FUNCTION_BLOCK FB_ProfidriveGSM_Test EXTENDS TcUnit.FB_TestSuite

TestState_S0();
TestState_S1();
TestState_S2();
TestState_S3();
TestState_S4();
TestState_S51();
TestState_S52();

TestTransitions_S0();
TestTransitions_S1();
TestTransitions_S2();
TestTransitions_S3();
TestTransitions_S4();
TestTransitions_S51();
TestTransitions_S52();

METHOD TestState_S0 : BOOL
VAR
	fbFSM 				: FB_ProfidriveGSM;
	stStatusExpected	: ST_ProfidriveGSM_Status;
END_VAR
TEST('Set State S0');

//Arrange
fbFSM.eState := E_ProfidriveGSM_State.S0_Disabled;

stStatusExpected.b0_ReadyToSwitchOn 		:= FALSE;				
stStatusExpected.b1_ReadyForOperation 		:= FALSE;				
stStatusExpected.b2_OperationEnabled 		:= FALSE;
stStatusExpected.b6_SwitchingOnInhibited 	:= FALSE;

//Act
fbFSM();

//Assert

AssertEquals_BOOL(stStatusExpected.b0_ReadyToSwitchOn, fbFSM.nStatus.b0_ReadyToSwitchOn, 'b0_ReadyToSwitchOn: AssertEquals not returning expected value');
AssertEquals_BOOL(stStatusExpected.b1_ReadyForOperation, fbFSM.nStatus.b1_ReadyForOperation, 'b1_ReadyForOperation: AssertEquals not returning expected value');
AssertEquals_BOOL(stStatusExpected.b2_OperationEnabled, fbFSM.nStatus.b2_OperationEnabled, 'b2_OperationEnabled: AssertEquals not returning expected value');	
AssertEquals_BOOL(stStatusExpected.b6_SwitchingOnInhibited, fbFSM.nStatus.b6_SwitchingOnInhibited, 'b6_SwitchingOnInhibited: AssertEquals not returning expected value');	

TEST_FINISHED();
END_METHOD

METHOD TestState_S1 : BOOL
VAR
	fbFSM 				: FB_ProfidriveGSM;
	stStatusExpected	: ST_ProfidriveGSM_Status;
END_VAR
TEST('Set State S1');

//Arrange
fbFSM.eState := E_ProfidriveGSM_State.S1_SwitchingOnInhibited;

stStatusExpected.b0_ReadyToSwitchOn 		:= FALSE;				
stStatusExpected.b1_ReadyForOperation 		:= FALSE;				
stStatusExpected.b2_OperationEnabled 		:= FALSE;
stStatusExpected.b6_SwitchingOnInhibited 	:= TRUE;

//Act
fbFSM();

//Assert
AssertEquals_BOOL(stStatusExpected.b0_ReadyToSwitchOn, fbFSM.nStatus.b0_ReadyToSwitchOn, 'b0_ReadyToSwitchOn: AssertEquals not returning expected value');
AssertEquals_BOOL(stStatusExpected.b1_ReadyForOperation, fbFSM.nStatus.b1_ReadyForOperation, 'b1_ReadyForOperation: AssertEquals not returning expected value');
AssertEquals_BOOL(stStatusExpected.b2_OperationEnabled, fbFSM.nStatus.b2_OperationEnabled, 'b2_OperationEnabled: AssertEquals not returning expected value');	
AssertEquals_BOOL(stStatusExpected.b6_SwitchingOnInhibited, fbFSM.nStatus.b6_SwitchingOnInhibited, 'b6_SwitchingOnInhibited: AssertEquals not returning expected value');	

TEST_FINISHED();
END_METHOD

METHOD TestState_S2 : BOOL
VAR
	fbFSM 				: FB_ProfidriveGSM;
	stStatusExpected	: ST_ProfidriveGSM_Status;
END_VAR
TEST('Set State S2');

//Arrange
fbFSM.eState := E_ProfidriveGSM_State.S2_ReadyForSwitchingOn;

stStatusExpected.b0_ReadyToSwitchOn 		:= TRUE;				
stStatusExpected.b1_ReadyForOperation 		:= FALSE;				
stStatusExpected.b2_OperationEnabled 		:= FALSE;
stStatusExpected.b6_SwitchingOnInhibited 	:= FALSE;

//Act
fbFSM();

//Assert
AssertEquals_BOOL(stStatusExpected.b0_ReadyToSwitchOn, fbFSM.nStatus.b0_ReadyToSwitchOn, 'b0_ReadyToSwitchOn: AssertEquals not returning expected value');
AssertEquals_BOOL(stStatusExpected.b1_ReadyForOperation, fbFSM.nStatus.b1_ReadyForOperation, 'b1_ReadyForOperation: AssertEquals not returning expected value');
AssertEquals_BOOL(stStatusExpected.b2_OperationEnabled, fbFSM.nStatus.b2_OperationEnabled, 'b2_OperationEnabled: AssertEquals not returning expected value');	
AssertEquals_BOOL(stStatusExpected.b6_SwitchingOnInhibited, fbFSM.nStatus.b6_SwitchingOnInhibited, 'b6_SwitchingOnInhibited: AssertEquals not returning expected value');	

TEST_FINISHED();
END_METHOD

METHOD TestState_S3 : BOOL
VAR
	fbFSM 				: FB_ProfidriveGSM;
	stStatusExpected	: ST_ProfidriveGSM_Status;
END_VAR
TEST('Set State S3');

//Arrange
fbFSM.eState := E_ProfidriveGSM_State.S3_SwitchedOn;

stStatusExpected.b0_ReadyToSwitchOn 		:= TRUE;				
stStatusExpected.b1_ReadyForOperation 		:= TRUE;				
stStatusExpected.b2_OperationEnabled 		:= FALSE;
stStatusExpected.b6_SwitchingOnInhibited 	:= FALSE;

//Act
fbFSM();

//Assert
AssertEquals_BOOL(stStatusExpected.b0_ReadyToSwitchOn, fbFSM.nStatus.b0_ReadyToSwitchOn, 'b0_ReadyToSwitchOn: AssertEquals not returning expected value');
AssertEquals_BOOL(stStatusExpected.b1_ReadyForOperation, fbFSM.nStatus.b1_ReadyForOperation, 'b1_ReadyForOperation: AssertEquals not returning expected value');
AssertEquals_BOOL(stStatusExpected.b2_OperationEnabled, fbFSM.nStatus.b2_OperationEnabled, 'b2_OperationEnabled: AssertEquals not returning expected value');	
AssertEquals_BOOL(stStatusExpected.b6_SwitchingOnInhibited, fbFSM.nStatus.b6_SwitchingOnInhibited, 'b6_SwitchingOnInhibited: AssertEquals not returning expected value');	

TEST_FINISHED();
END_METHOD

METHOD TestState_S4 : BOOL
VAR
	fbFSM 				: FB_ProfidriveGSM;
	stStatusExpected	: ST_ProfidriveGSM_Status;
END_VAR
TEST('Set State S4');

//Arrange
fbFSM.eState := E_ProfidriveGSM_State.S4_Operation;

stStatusExpected.b0_ReadyToSwitchOn 		:= TRUE;				
stStatusExpected.b1_ReadyForOperation 		:= TRUE;				
stStatusExpected.b2_OperationEnabled 		:= TRUE;
stStatusExpected.b6_SwitchingOnInhibited 	:= FALSE;

//Act
fbFSM();

//Assert
AssertEquals_BOOL(stStatusExpected.b0_ReadyToSwitchOn, fbFSM.nStatus.b0_ReadyToSwitchOn, 'b0_ReadyToSwitchOn: AssertEquals not returning expected value');
AssertEquals_BOOL(stStatusExpected.b1_ReadyForOperation, fbFSM.nStatus.b1_ReadyForOperation, 'b1_ReadyForOperation: AssertEquals not returning expected value');
AssertEquals_BOOL(stStatusExpected.b2_OperationEnabled, fbFSM.nStatus.b2_OperationEnabled, 'b2_OperationEnabled: AssertEquals not returning expected value');	
AssertEquals_BOOL(stStatusExpected.b6_SwitchingOnInhibited, fbFSM.nStatus.b6_SwitchingOnInhibited, 'b6_SwitchingOnInhibited: AssertEquals not returning expected value');	

TEST_FINISHED();
END_METHOD

METHOD TestState_S51 : BOOL
VAR
	fbFSM 				: FB_ProfidriveGSM;
	stStatusExpected	: ST_ProfidriveGSM_Status;
END_VAR
TEST('Set State S51');

//Arrange
fbFSM.eState := E_ProfidriveGSM_State.S51_RampStop;

stStatusExpected.b0_ReadyToSwitchOn 		:= TRUE;				
stStatusExpected.b1_ReadyForOperation 		:= TRUE;				
stStatusExpected.b2_OperationEnabled 		:= FALSE;
stStatusExpected.b6_SwitchingOnInhibited 	:= FALSE;

//Act
fbFSM();

//Assert
AssertEquals_BOOL(stStatusExpected.b0_ReadyToSwitchOn, fbFSM.nStatus.b0_ReadyToSwitchOn, 'b0_ReadyToSwitchOn: AssertEquals not returning expected value');
AssertEquals_BOOL(stStatusExpected.b1_ReadyForOperation, fbFSM.nStatus.b1_ReadyForOperation, 'b1_ReadyForOperation: AssertEquals not returning expected value');
AssertEquals_BOOL(stStatusExpected.b2_OperationEnabled, fbFSM.nStatus.b2_OperationEnabled, 'b2_OperationEnabled: AssertEquals not returning expected value');	
AssertEquals_BOOL(stStatusExpected.b6_SwitchingOnInhibited, fbFSM.nStatus.b6_SwitchingOnInhibited, 'b6_SwitchingOnInhibited: AssertEquals not returning expected value');	

TEST_FINISHED();
END_METHOD

METHOD TestState_S52 : BOOL
VAR
	fbFSM 				: FB_ProfidriveGSM;
	stStatusExpected	: ST_ProfidriveGSM_Status;
END_VAR
TEST('Set State S52');

//Arrange
fbFSM.eState := E_ProfidriveGSM_State.S52_QuickStop;

stStatusExpected.b0_ReadyToSwitchOn 		:= TRUE;				
stStatusExpected.b1_ReadyForOperation 		:= TRUE;				
stStatusExpected.b2_OperationEnabled 		:= FALSE;
stStatusExpected.b6_SwitchingOnInhibited 	:= FALSE;

//Act
fbFSM();

//Assert
AssertEquals_BOOL(stStatusExpected.b0_ReadyToSwitchOn, fbFSM.nStatus.b0_ReadyToSwitchOn, 'b0_ReadyToSwitchOn: AssertEquals not returning expected value');
AssertEquals_BOOL(stStatusExpected.b1_ReadyForOperation, fbFSM.nStatus.b1_ReadyForOperation, 'b1_ReadyForOperation: AssertEquals not returning expected value');
AssertEquals_BOOL(stStatusExpected.b2_OperationEnabled, fbFSM.nStatus.b2_OperationEnabled, 'b2_OperationEnabled: AssertEquals not returning expected value');	
AssertEquals_BOOL(stStatusExpected.b6_SwitchingOnInhibited, fbFSM.nStatus.b6_SwitchingOnInhibited, 'b6_SwitchingOnInhibited: AssertEquals not returning expected value');	

TEST_FINISHED();
END_METHOD

METHOD TestTransitions_S0 : BOOL
VAR
	fbFSM 				: FB_ProfidriveGSM;
	stStatusExpected	: ST_ProfidriveGSM_Status;
	nStatusExpected 	: WORD;
END_VAR
TEST('Transition S0>S0');

//Arrange
fbFSM.bPowerOn := FALSE;
fbFSM.eState := E_ProfidriveGSM_State.S0_Disabled;

//Act
fbFSM();

//Assert
AssertEquals_INT(E_ProfidriveGSM_State.S0_Disabled, fbFSM.eState, 'eState: AssertEquals not returning expected value');

TEST_FINISHED();


TEST('Transition S0>S1');

//Arrange
fbFSM.bPowerOn := TRUE;
fbFSM.eState := E_ProfidriveGSM_State.S0_Disabled;

//Act
fbFSM();

//Assert
AssertEquals_INT(E_ProfidriveGSM_State.S1_SwitchingOnInhibited, fbFSM.eState, 'eState: AssertEquals not returning expected value');

TEST_FINISHED();
END_METHOD

METHOD TestTransitions_S1 : BOOL
VAR
	fbFSM 				: FB_ProfidriveGSM;
	stStatusExpected	: ST_ProfidriveGSM_Status;
	nStatusExpected 	: WORD;
END_VAR
TEST('Transition S1>S2');

//Arrange
fbFSM.bPowerOn := TRUE;
fbFSM.eState := E_ProfidriveGSM_State.S1_SwitchingOnInhibited;

fbFSM.nControl.b0_On 				:= FALSE;
fbFSM.nControl.b1_CoastStop 		:= TRUE;
fbFSM.nControl.b2_QuickStop 		:= TRUE;

//Act
fbFSM();

//Assert
AssertEquals_INT(E_ProfidriveGSM_State.S2_ReadyForSwitchingOn, fbFSM.eState, 'eState: AssertEquals not returning expected value');

TEST_FINISHED();
END_METHOD

METHOD TestTransitions_S2 : BOOL
VAR
	fbFSM 				: FB_ProfidriveGSM;
	stStatusExpected	: ST_ProfidriveGSM_Status;
	nStatusExpected 	: WORD;
END_VAR
TEST('Transition S2>S1 Case_1');

//Arrange
fbFSM.bPowerOn := TRUE;
fbFSM.eState := E_ProfidriveGSM_State.S2_ReadyForSwitchingOn;

fbFSM.nControl.b0_On 				:= TRUE;
fbFSM.nControl.b1_CoastStop 		:= FALSE;
fbFSM.nControl.b2_QuickStop 		:= TRUE;

//Act
fbFSM();

//Assert
AssertEquals_INT(E_ProfidriveGSM_State.S1_SwitchingOnInhibited, fbFSM.eState, 'eState: AssertEquals not returning expected value');

TEST_FINISHED();


TEST('Transition S2>S1 Case_2');

//Arrange
fbFSM.bPowerOn := TRUE;
fbFSM.eState := E_ProfidriveGSM_State.S2_ReadyForSwitchingOn;

fbFSM.nControl.b0_On 				:= TRUE;
fbFSM.nControl.b1_CoastStop 		:= TRUE;
fbFSM.nControl.b2_QuickStop 		:= FALSE;

//Act
fbFSM();

//Assert
AssertEquals_INT(E_ProfidriveGSM_State.S1_SwitchingOnInhibited, fbFSM.eState, 'eState: AssertEquals not returning expected value');

TEST_FINISHED();


TEST('Transition S2 Still');

//Arrange
fbFSM.bPowerOn := TRUE;
fbFSM.eState := E_ProfidriveGSM_State.S2_ReadyForSwitchingOn;

fbFSM.nControl.b0_On 				:= FALSE;
fbFSM.nControl.b1_CoastStop 		:= TRUE;
fbFSM.nControl.b2_QuickStop 		:= TRUE;

//Act
fbFSM();

//Assert
AssertEquals_INT(E_ProfidriveGSM_State.S2_ReadyForSwitchingOn, fbFSM.eState, 'eState: AssertEquals not returning expected value');

TEST_FINISHED();


TEST('Transition S2>S3');

//Arrange
fbFSM.bPowerOn := TRUE;
fbFSM.eState := E_ProfidriveGSM_State.S2_ReadyForSwitchingOn;

fbFSM.nControl.b0_On 				:= TRUE;
fbFSM.nControl.b1_CoastStop 		:= TRUE;
fbFSM.nControl.b2_QuickStop 		:= TRUE;

//Act
fbFSM();

//Assert
AssertEquals_INT(E_ProfidriveGSM_State.S3_SwitchedOn, fbFSM.eState, 'eState: AssertEquals not returning expected value');

TEST_FINISHED();
END_METHOD

METHOD TestTransitions_S3 : BOOL
VAR
	fbFSM 				: FB_ProfidriveGSM;
	stStatusExpected	: ST_ProfidriveGSM_Status;
	nStatusExpected 	: WORD;
END_VAR
TEST('Transition S3>S1 Case_1');

//Arrange
fbFSM.bPowerOn := TRUE;
fbFSM.eState := E_ProfidriveGSM_State.S3_SwitchedOn;

fbFSM.nControl.b0_On 				:= TRUE;
fbFSM.nControl.b1_CoastStop 		:= FALSE;
fbFSM.nControl.b2_QuickStop 		:= TRUE;

//Act
fbFSM();

//Assert
AssertEquals_INT(E_ProfidriveGSM_State.S1_SwitchingOnInhibited, fbFSM.eState, 'eState: AssertEquals not returning expected value');

TEST_FINISHED();


TEST('Transition S3>S1 Case_2');

//Arrange
fbFSM.bPowerOn := TRUE;
fbFSM.eState := E_ProfidriveGSM_State.S3_SwitchedOn;

fbFSM.nControl.b0_On 				:= TRUE;
fbFSM.nControl.b1_CoastStop 		:= TRUE;
fbFSM.nControl.b2_QuickStop 		:= FALSE;

//Act
fbFSM();

//Assert
AssertEquals_INT(E_ProfidriveGSM_State.S1_SwitchingOnInhibited, fbFSM.eState, 'eState: AssertEquals not returning expected value');

TEST_FINISHED();


TEST('Transition S3 Still');

//Arrange
fbFSM.bPowerOn := TRUE;
fbFSM.eState := E_ProfidriveGSM_State.S3_SwitchedOn;

fbFSM.nControl.b0_On 				:= TRUE;
fbFSM.nControl.b1_CoastStop 		:= TRUE;
fbFSM.nControl.b2_QuickStop 		:= TRUE;
fbFSM.nControl.b3_EnableOperation  := FALSE;

//Act
fbFSM();

//Assert
AssertEquals_INT(E_ProfidriveGSM_State.S3_SwitchedOn, fbFSM.eState, 'eState: AssertEquals not returning expected value');

TEST_FINISHED();


TEST('Transition S3>S2');

//Arrange
fbFSM.bPowerOn := TRUE;
fbFSM.eState := E_ProfidriveGSM_State.S3_SwitchedOn;

fbFSM.nControl.b0_On 				:= FALSE;
fbFSM.nControl.b1_CoastStop 		:= TRUE;
fbFSM.nControl.b2_QuickStop 		:= TRUE;

//Act
fbFSM();

//Assert
AssertEquals_INT(E_ProfidriveGSM_State.S2_ReadyForSwitchingOn, fbFSM.eState, 'eState: AssertEquals not returning expected value');

TEST_FINISHED();


TEST('Transition S3>S4');

//Arrange
fbFSM.bPowerOn := TRUE;
fbFSM.eState := E_ProfidriveGSM_State.S3_SwitchedOn;

fbFSM.nControl.b0_On 				:= TRUE;
fbFSM.nControl.b1_CoastStop 		:= TRUE;
fbFSM.nControl.b2_QuickStop 		:= TRUE;
fbFSM.nControl.b3_EnableOperation  := TRUE;

//Act
fbFSM();

//Assert
AssertEquals_INT(E_ProfidriveGSM_State.S4_Operation, fbFSM.eState, 'eState: AssertEquals not returning expected value');

TEST_FINISHED();
END_METHOD

METHOD TestTransitions_S4 : BOOL
VAR
	fbFSM 				: FB_ProfidriveGSM;
	stStatusExpected	: ST_ProfidriveGSM_Status;
	nStatusExpected 	: WORD;
END_VAR
TEST('Transition S4>S1');

//Arrange
fbFSM.bPowerOn := TRUE;
fbFSM.eState := E_ProfidriveGSM_State.S4_Operation;

fbFSM.nControl.b0_On 				:= FALSE;
fbFSM.nControl.b1_CoastStop 		:= FALSE;
fbFSM.nControl.b2_QuickStop 		:= FALSE;

//Act
fbFSM();

//Assert
AssertEquals_INT(E_ProfidriveGSM_State.S1_SwitchingOnInhibited, fbFSM.eState, 'eState: AssertEquals not returning expected value');

TEST_FINISHED();


TEST('Transition S4>S52');

//Arrange
fbFSM.bPowerOn := TRUE;
fbFSM.eState := E_ProfidriveGSM_State.S4_Operation;

fbFSM.nControl.b0_On 				:= FALSE;
fbFSM.nControl.b1_CoastStop 		:= TRUE;
fbFSM.nControl.b2_QuickStop 		:= FALSE;

//Act
fbFSM();

//Assert
AssertEquals_INT(E_ProfidriveGSM_State.S52_QuickStop, fbFSM.eState, 'eState: AssertEquals not returning expected value');

TEST_FINISHED();


TEST('Transition S4>S51');

//Arrange
fbFSM.bPowerOn := TRUE;
fbFSM.eState := E_ProfidriveGSM_State.S4_Operation;

fbFSM.nControl.b0_On 				:= FALSE;
fbFSM.nControl.b1_CoastStop 		:= TRUE;
fbFSM.nControl.b2_QuickStop 		:= TRUE;
fbFSM.nControl.b3_EnableOperation 	:= FALSE;

//Act
fbFSM();

//Assert
AssertEquals_INT(E_ProfidriveGSM_State.S51_RampStop, fbFSM.eState, 'eState: AssertEquals not returning expected value');

TEST_FINISHED();


TEST('Transition S4>S3');

//Arrange
fbFSM.bPowerOn := TRUE;
fbFSM.eState := E_ProfidriveGSM_State.S4_Operation;

fbFSM.nControl.b0_On 				:= TRUE;
fbFSM.nControl.b1_CoastStop 		:= TRUE;
fbFSM.nControl.b2_QuickStop 		:= TRUE;
fbFSM.nControl.b3_EnableOperation 	:= FALSE;

//Act
fbFSM();

//Assert
AssertEquals_INT(E_ProfidriveGSM_State.S3_SwitchedOn, fbFSM.eState, 'eState: AssertEquals not returning expected value');

TEST_FINISHED();
END_METHOD

METHOD TestTransitions_S51 : BOOL
VAR
	fbFSM 				: FB_ProfidriveGSM;
	stStatusExpected	: ST_ProfidriveGSM_Status;
	nStatusExpected 	: WORD;
END_VAR
TEST('Transition S51 Still');

//Arrange
fbFSM.bPowerOn := TRUE;
fbFSM.eState := E_ProfidriveGSM_State.S51_RampStop;

fbFSM.bStandstill					:= FALSE;
fbFSM.nControl.b0_On 				:= FALSE;
fbFSM.nControl.b1_CoastStop 		:= TRUE;
fbFSM.nControl.b2_QuickStop 		:= TRUE;
fbFSM.nControl.b3_EnableOperation 	:= TRUE;

//Act
fbFSM();

//Assert
AssertEquals_INT(E_ProfidriveGSM_State.S51_RampStop, fbFSM.eState, 'eState: AssertEquals not returning expected value');

TEST_FINISHED();


TEST('Transition S51>S1');

//Arrange
fbFSM.bPowerOn := TRUE;
fbFSM.eState := E_ProfidriveGSM_State.S51_RampStop;

fbFSM.bStandstill					:= FALSE;
fbFSM.nControl.b0_On 				:= FALSE;
fbFSM.nControl.b1_CoastStop 		:= FALSE;
fbFSM.nControl.b2_QuickStop 		:= FALSE;
fbFSM.nControl.b3_EnableOperation 	:= FALSE;

//Act
fbFSM();

//Assert
AssertEquals_INT(E_ProfidriveGSM_State.S1_SwitchingOnInhibited, fbFSM.eState, 'eState: AssertEquals not returning expected value');

TEST_FINISHED();


TEST('Transition S51>S52');

//Arrange
fbFSM.bPowerOn := TRUE;
fbFSM.eState := E_ProfidriveGSM_State.S51_RampStop;

fbFSM.bStandstill					:= FALSE;
fbFSM.nControl.b0_On 				:= FALSE;
fbFSM.nControl.b1_CoastStop 		:= TRUE;
fbFSM.nControl.b2_QuickStop 		:= FALSE;
fbFSM.nControl.b3_EnableOperation 	:= TRUE;

//Act
fbFSM();

//Assert
AssertEquals_INT(E_ProfidriveGSM_State.S52_QuickStop, fbFSM.eState, 'eState: AssertEquals not returning expected value');

TEST_FINISHED();


TEST('Transition S51>S2 Case_1');

//Arrange
fbFSM.bPowerOn := TRUE;
fbFSM.eState := E_ProfidriveGSM_State.S51_RampStop;

fbFSM.bStandstill					:= FALSE;
fbFSM.nControl.b0_On 				:= FALSE;
fbFSM.nControl.b1_CoastStop 		:= TRUE;
fbFSM.nControl.b2_QuickStop 		:= TRUE;
fbFSM.nControl.b3_EnableOperation 	:= FALSE;

//Act
fbFSM();

//Assert
AssertEquals_INT(E_ProfidriveGSM_State.S2_ReadyForSwitchingOn, fbFSM.eState, 'eState: AssertEquals not returning expected value');

TEST_FINISHED();


TEST('Transition S51>S2 Case_2');

//Arrange
fbFSM.bPowerOn := TRUE;
fbFSM.eState := E_ProfidriveGSM_State.S51_RampStop;

fbFSM.bStandstill					:= TRUE;
fbFSM.nControl.b0_On 				:= FALSE;
fbFSM.nControl.b1_CoastStop 		:= TRUE;
fbFSM.nControl.b2_QuickStop 		:= TRUE;
fbFSM.nControl.b3_EnableOperation 	:= TRUE;

//Act
fbFSM();

//Assert
AssertEquals_INT(E_ProfidriveGSM_State.S2_ReadyForSwitchingOn, fbFSM.eState, 'eState: AssertEquals not returning expected value');

TEST_FINISHED();


TEST('Transition S51>S4');

//Arrange
fbFSM.bPowerOn := TRUE;
fbFSM.eState := E_ProfidriveGSM_State.S51_RampStop;

fbFSM.bStandstill					:= FALSE;
fbFSM.nControl.b0_On 				:= TRUE;
fbFSM.nControl.b1_CoastStop 		:= TRUE;
fbFSM.nControl.b2_QuickStop 		:= TRUE;
fbFSM.nControl.b3_EnableOperation 	:= TRUE;

//Act
fbFSM();

//Assert
AssertEquals_INT(E_ProfidriveGSM_State.S4_Operation, fbFSM.eState, 'eState: AssertEquals not returning expected value');

TEST_FINISHED();
END_METHOD

METHOD TestTransitions_S52 : BOOL
VAR
	fbFSM 				: FB_ProfidriveGSM;
	stStatusExpected	: ST_ProfidriveGSM_Status;
	nStatusExpected 	: WORD;
END_VAR
TEST('Transition S52 Still');

//Arrange
fbFSM.bPowerOn := TRUE;
fbFSM.eState := E_ProfidriveGSM_State.S52_QuickStop;

fbFSM.bStandstill					:= FALSE;
fbFSM.nControl.b0_On 				:= FALSE;
fbFSM.nControl.b1_CoastStop 		:= TRUE;
fbFSM.nControl.b2_QuickStop 		:= FALSE;
fbFSM.nControl.b3_EnableOperation 	:= TRUE;

//Act
fbFSM();

//Assert
AssertEquals_INT(E_ProfidriveGSM_State.S52_QuickStop, fbFSM.eState, 'eState: AssertEquals not returning expected value');

TEST_FINISHED();


TEST('Transition S51>S1 Case_1');

//Arrange
fbFSM.bPowerOn := TRUE;
fbFSM.eState := E_ProfidriveGSM_State.S52_QuickStop;

fbFSM.bStandstill					:= FALSE;
fbFSM.nControl.b0_On 				:= FALSE;
fbFSM.nControl.b1_CoastStop 		:= FALSE;
fbFSM.nControl.b2_QuickStop 		:= FALSE;
fbFSM.nControl.b3_EnableOperation 	:= FALSE;

//Act
fbFSM();

//Assert
AssertEquals_INT(E_ProfidriveGSM_State.S1_SwitchingOnInhibited, fbFSM.eState, 'eState: AssertEquals not returning expected value');

TEST_FINISHED();


TEST('Transition S52>S1 Case_2');

//Arrange
fbFSM.bPowerOn := TRUE;
fbFSM.eState := E_ProfidriveGSM_State.S52_QuickStop;

fbFSM.bStandstill					:= FALSE;
fbFSM.nControl.b0_On 				:= FALSE;
fbFSM.nControl.b1_CoastStop 		:= TRUE;
fbFSM.nControl.b2_QuickStop 		:= FALSE;
fbFSM.nControl.b3_EnableOperation 	:= FALSE;

//Act
fbFSM();

//Assert
AssertEquals_INT(E_ProfidriveGSM_State.S1_SwitchingOnInhibited, fbFSM.eState, 'eState: AssertEquals not returning expected value');

TEST_FINISHED();

TEST('Transition S52>S1 Case_3');

//Arrange
fbFSM.bPowerOn := TRUE;
fbFSM.eState := E_ProfidriveGSM_State.S52_QuickStop;

fbFSM.bStandstill					:= TRUE;
fbFSM.nControl.b0_On 				:= FALSE;
fbFSM.nControl.b1_CoastStop 		:= TRUE;
fbFSM.nControl.b2_QuickStop 		:= FALSE;
fbFSM.nControl.b3_EnableOperation 	:= TRUE;

//Act
fbFSM();

//Assert
AssertEquals_INT(E_ProfidriveGSM_State.S1_SwitchingOnInhibited, fbFSM.eState, 'eState: AssertEquals not returning expected value');

TEST_FINISHED();
END_METHOD

END_FUNCTION_BLOCK

(* stored: Version 1.1.0.1, ProductVersion 3.1.4024.12
   POU FB_ProfidriveGSM_Test: Id {f35b0c2b-bf7b-08eb-1441-1129517b119a}, SpecialFunc None
   Method TestState_S0: Id {0722bab6-5316-0ca8-2a8f-9bc8f87e4ce0}
   Method TestState_S1: Id {21e4e4c6-7feb-0913-2530-a3403cbcc57a}
   Method TestState_S2: Id {4fb6cd64-4731-0227-14fa-4933a49e4a58}
   Method TestState_S3: Id {c3cc8a49-e00d-0a3c-0091-1a9173012426}
   Method TestState_S4: Id {eb2efc53-7797-0db0-0d46-8c839adaf33d}
   Method TestState_S51: Id {cfba5483-0838-003a-2805-865bb90498ab}
   Method TestState_S52: Id {945fa724-fc62-048e-1192-5818b8a722a4}
   Method TestTransitions_S0: Id {2cf2b562-f51d-0d29-3dc8-40331aa2da09}
   Method TestTransitions_S1: Id {2a966d2a-86e5-0a57-19ef-7d9154ededd2}
   Method TestTransitions_S2: Id {45938320-5191-0c9a-0945-99084c0adb67}
   Method TestTransitions_S3: Id {e6c30110-0cba-0a05-3236-ecfd0aa2490c}
   Method TestTransitions_S4: Id {ce52dda4-01c8-0635-35d0-2b4cc0c49e96}
   Method TestTransitions_S51: Id {03057e99-f4d5-0ba5-2481-acd61d83d47a}
   Method TestTransitions_S52: Id {d39f8d13-3865-039d-1f75-63bbcd8add6e} *)
